{attribute 'qualified_only'}
VAR_GLOBAL
    Axis1 : ST_AxisInternalSts;   // PLC 内部使用：功能块详细状态
END_VAR

(* stored: Version 1.1.0.1, ProductVersion 3.1.4026.18
   GVL GVL_AxisInternal: Id {08854f79-8ee8-4b81-9a66-4319a5412a32} *)
